# EPICS autosave request: laudaRE2xx/lRE2xx_settings.req
$(P):DISABLE
$(P):RRATE
$(P):RTEMP
$(P):SET_PUMP
$(P):SET_TEMP
